FUNCTION_BLOCK GreenMasterSmokeControl_Base
VAR_IN_OUT
	Parameters: GreenMasterBaseParameters;	
	ParametersSC: SmokeControlParametersBase;
END_VAR
VAR_INPUT
	EN: BOOL;
END_VAR
VAR_OUTPUT
	FireAlarm: BOOL;
END_VAR
VAR
END_VAR

END_FUNCTION_BLOCK

(* stored: Version 1.1.0.1, ProductVersion 3.1.4024.6
   POU GreenMasterSmokeControl_Base: Id {f0a50325-de03-4659-be38-0d5b55dfc595}, SpecialFunc None *)
